% RSLogix 500 project TIMER IN LADDER LOGIC_BAK006.RSS, saved by version 8.30.00.16 %
PROJECT "UNTITLED"    % processor: Bul.1763 MicroLogix 1100 Series B %

PROGRAM FILES
  LAD 2   5 rungs

DATA FILES
  O0 OUTPUT  4 elements
  I1 INPUT  6 elements
  S2 STATUS  66 elements
  B3 BINARY  1 elements
  T4 TIMER  1 elements
  C5 COUNTER  1 elements
  R6 CONTROL  1 elements
  N7 INTEGER  1 elements
  F8 FLOAT  1 elements

LADDER 2
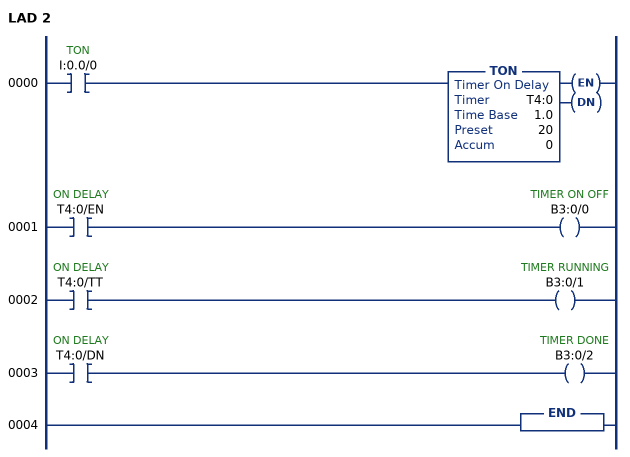
% Rung: 0 %
SOR XIC I:0.0/0 TON T4:0 1.0 20 0 EOR
%   I:0.0/0  TON %
% Rung: 1 %
SOR XIC T4:0/EN OTE B3:0/0 EOR
%   T4:0/EN  "ON DELAY" %
%   B3:0/0  "TIMER ON OFF" %
% Rung: 2 %
SOR XIC T4:0/TT OTE B3:0/1 EOR
%   T4:0/TT  "ON DELAY" %
%   B3:0/1  "TIMER RUNNING" %
% Rung: 3 %
SOR XIC T4:0/DN OTE B3:0/2 EOR
%   T4:0/DN  "ON DELAY" %
%   B3:0/2  "TIMER DONE" %
% Rung: 4 %
SOR END EOR

DATA TABLE (non-zero values as saved)
DATA T4
% .PRE .ACC %
% T4:0 % 20 0
